Staubli VAL3: loadCycle.pgx

public program loadCycle(string x_sItem, num& x_nResult[])
  local string l_sType
  local string l_sPath
begin
  // load the select trajectory..already loaded
  call getTrajType(l_sType)
  if find(pt:libPath(),saveData:sPathTraj)==-1
    pt:libLoad(saveData:sPathTraj+l_sType)
    delay(0)
  endIf
  if isDefined(pt:tTraj[x_sItem])
    // use the type...
    call pt:link_it(x_sItem)
    sTrajCycle=x_sItem
  else
    x_nResult=-1
  endIf
end
